// TwinCAT 3 PLC project STRIX1200
// ProgramVersion: 3.1.4024.0
// libraries:
//   CmpBitmapPool, * (System)
//   Tc2_MC2, * (Beckhoff Automation GmbH)
//   Tc2_Standard, * (Beckhoff Automation GmbH)
//   Tc2_System, * (Beckhoff Automation GmbH)
//   Tc2_Utilities, * (Beckhoff Automation GmbH)
//   Tc3_Module, * (Beckhoff Automation GmbH)
//   VisuDialogs, * (System)
// project tree:
//   / GlobalTextList.TcGTLO, PlcTask.TcTTO, Visualization Manager.TcVMO (not stored), VISU_TASK.TcTTO
//   POUs/ACTION/ E_ACTION_STATE.TcDUT, FB_ACTION.TcPOU (not stored), FB_AnalogSensor.TcPOU (not stored), vACTION.TcVIS
//   POUs/AXES/ AXES_CYCLE.TcPOU, E_AXIS_STATE.TcDUT, FB_Axis.TcPOU, GVL_AXES.TcGVL, vAXES2.TcVIS, vAXIS.TcVIS, vAXES1.TcVIS
//   POUs/EVENT_LOGGER/ E_EventType.TcDUT, FB_EventLogger.TcPOU, GVL_EVENT_LOGGER.TcGVL, ST_Event.TcDUT, UpdateEventTimestampWithSystemTime.TcPOU, UpdateTimeStamp.TcPOU, vEVENT_LOGGER.TcVIS
//   POUs/ GVL_MAIN.TcGVL (not stored), MAIN.TcPOU (not stored)
//   POUs/IOs/ sEL1809.TcDUT, sEL2809.TcDUT
//   POUs/PISTONS/ E_PISTON_STATE.TcDUT, E_PISTON_TYPE.TcDUT, FB_PISTON.TcPOU, PIST_CYCLE.TcPOU, ST_PISTON.TcDUT, vPISTONS.TcVIS, vPISTON.TcVIS
//   VISUs/VISUs/ ImagePool.TcIPO (not stored), vCOMM.TcVIS, vMAIN.TcVIS
// real-time tasks:
//   TASK PlcTask: cycle T#10ms, priority 20, ADS port 350
//   TASK VISU_TASK: cycle T#70000us, priority 30, ADS port 351
// motion (NC):
//   TASK NC-Task 1 SAF: cycle T#2ms, priority 4, ADS port 501
//   TASK NC-Task 1 SVB: cycle T#10ms, priority 8, ADS port 511
//   AXIS XY1 (id 2)
//     Dynamic: AccelerationMaximum=1500, DecelerationMaximum=1500, Acceleration=400, Deceleration=400, Jerk=40000
//     Velo: SlowManual=3, FastManual=6, Maximum=200
//     OtherSettings: AllowMotionCmdToSlave=true
//     encoder EncType=4
//       EncPara: ScaleFactorNumerator=0.001, EncMode=3, MaxCount=#xffffffff
//         TimeComp: TimeCompMode=1, EncDelayCycles=4
//     drive DrvType=5
//       Analog: VeloReferenz=200, TorqueSetpointScale=10, ScaleFactorActTorque=0.1
//       TimeComp: TimeCompMode=1, TaskDelayCycles=1
//     controller CtrType=1
//       CtrPara: PriorControlFactor=1
//         PosDiffControl: Enable=false
//         PID: PosKp=50
//         Observer: BandWidth=20
//   AXIS LIFT2 (id 3)
//     OtherSettings: AllowMotionCmdToSlave=true
//     encoder EncType=1
//     drive DrvType=5
//       Analog: TorqueSetpointScale=10, ScaleFactorActTorque=0.1
//       TimeComp: TaskDelayCycles=1
//     controller CtrType=1
//       CtrPara: PriorControlFactor=1
//         PID: PosKp=50
//         Observer: BandWidth=20
//   AXIS XY2 (id 4)
//     OtherSettings: AllowMotionCmdToSlave=true
//     encoder EncType=1
//     drive DrvType=5
//       Analog: TorqueSetpointScale=10, ScaleFactorActTorque=0.1
//       TimeComp: TaskDelayCycles=1
//     controller CtrType=1
//       CtrPara: PriorControlFactor=1
//         PID: PosKp=50
//         Observer: BandWidth=20
//   AXIS LIFT1 (id 1)
//     Dynamic: AccelerationMaximum=300, DecelerationMaximum=300, Acceleration=400, Deceleration=400, Jerk=40000
//     Velo: SlowManual=10, FastManual=30, Maximum=200
//     OtherSettings: AllowMotionCmdToSlave=true
//     encoder EncType=4
//       EncPara: ScaleFactorNumerator=0.001, EncMode=3, MaxCount=#xffffffff
//         TimeComp: TimeCompMode=1
//     drive DrvType=5
//       Analog: VeloReferenz=200, TorqueSetpointScale=10, ScaleFactorActTorque=0.1
//       TimeComp: TimeCompMode=1, TaskDelayCycles=1
//     controller CtrType=1
//       CtrPara: PriorControlFactor=1
//         PosDiffControl: Enable=false
//         PID: PosKp=50
//         Observer: BandWidth=20
// I/O:
//   DEVICE Device 1 (EtherCAT), AmsNetId 5.144.185.120.2.1
//     Term 1 (EK1100) [EK1100 EtherCAT Coupler (2A E-Bus)]
//       Term 2 (EL1809) [EL1809 16Ch. Dig. Input 24V, 3ms]
//       Term 3 (EL2809) [EL2809 16Ch. Dig. Output 24V, 0.5A]
//       Term 4 (EL2522) [EL2522 2Ch. Pulse Train Output]
//       Term 5 (EL3064) [EL3064 4Ch. Ana. Input 0-10V]
//       Term 6 (EL9011) [EL9011 End Terminal]
// variable links:
//   NC-Task 1 SAF/Axes/LIFT1 <-> Device 1 (EtherCAT)/Term 1 (EK1100)/Term 4 (EL2522)
//     Drive/Inputs/In/nDcOutputTime <-> InfoData/DcOutputShift
//     Drive/Inputs/In/nState1 @bit 6 <-> PTO Status Channel 2/Status/Error
//     Drive/Inputs/In/nState1 @bit 1 <-> PTO Status Channel 2/Status/Ramp active
//     Drive/Inputs/In/nState1 <-> PTO Status Channel 2/Status/Sel. Ack/End counter
//     Drive/Inputs/In/nState2 @bit 5 <-> PTO Status Channel 2/Status/Sync error
//     Drive/Inputs/In/nState2 @bit 7 <-> PTO Status Channel 2/Status/TxPDO Toggle
//     Drive/Inputs/In/nState4 @bit 1 <-> WcState/InputToggle
//     Drive/Inputs/In/nState4 <-> WcState/WcState
//     Drive/Outputs/Out/nCtrl1 @bit 1 <-> PTO Control Channel 2/Control/Disable ramp
//     Drive/Outputs/Out/nCtrl1 <-> PTO Control Channel 2/Control/Frequency select
//     Drive/Outputs/Out/nCtrl1 @bit 2 <-> PTO Control Channel 2/Control/Go counter
//     Drive/Outputs/Out/nDataOut1[0] <-> PTO Control Channel 2/Frequency value
//     Drive/Outputs/Out/nDataOut5 <-> PTO Target Channel 2/Target counter value
//     Enc/Inputs/In/nDataIn1 <-> ENC Status Channel 2/Counter value
//     Enc/Inputs/In/nDcInputTime <-> InfoData/DcInputShift
//     Enc/Inputs/In/nState1 @bit 4 <-> ENC Status Channel 2/Status/Counter overflow
//     Enc/Inputs/In/nState1 @bit 3 <-> ENC Status Channel 2/Status/Counter underflow
//     Enc/Inputs/In/nState1 @bit 2 <-> ENC Status Channel 2/Status/Set counter done
//     Enc/Inputs/In/nState2 @bit 5 <-> ENC Status Channel 2/Status/Sync error
//     Enc/Inputs/In/nState2 @bit 6 <-> ENC Status Channel 2/Status/TxPDO State
//     Enc/Inputs/In/nState2 @bit 7 <-> ENC Status Channel 2/Status/TxPDO Toggle
//     Enc/Inputs/In/nState4 @bit 1 <-> WcState/InputToggle
//     Enc/Inputs/In/nState4 <-> WcState/WcState
//     Enc/Outputs/Out/nCtrl1 @bit 2 <-> ENC Control Channel 2/Control/Set counter
//     Enc/Outputs/Out/nCtrl2 @bit 7 <-> ENC Control Channel 2/Control/Reserved
//     Enc/Outputs/Out/nDataOut1 <-> ENC Control Channel 2/Set counter value
//   NC-Task 1 SAF/Axes/XY1 <-> Device 1 (EtherCAT)/Term 1 (EK1100)/Term 4 (EL2522)
//     Drive/Inputs/In/nDcOutputTime <-> InfoData/DcOutputShift
//     Drive/Inputs/In/nState1 @bit 6 <-> PTO Status Channel 1/Status/Error
//     Drive/Inputs/In/nState1 @bit 1 <-> PTO Status Channel 1/Status/Ramp active
//     Drive/Inputs/In/nState1 <-> PTO Status Channel 1/Status/Sel. Ack/End counter
//     Drive/Inputs/In/nState2 @bit 5 <-> PTO Status Channel 1/Status/Sync error
//     Drive/Inputs/In/nState2 @bit 7 <-> PTO Status Channel 1/Status/TxPDO Toggle
//     Drive/Inputs/In/nState4 @bit 1 <-> WcState/InputToggle
//     Drive/Inputs/In/nState4 <-> WcState/WcState
//     Drive/Outputs/Out/nCtrl1 @bit 1 <-> PTO Control Channel 1/Control/Disable ramp
//     Drive/Outputs/Out/nCtrl1 <-> PTO Control Channel 1/Control/Frequency select
//     Drive/Outputs/Out/nCtrl1 @bit 2 <-> PTO Control Channel 1/Control/Go counter
//     Drive/Outputs/Out/nDataOut1[0] <-> PTO Control Channel 1/Frequency value
//     Drive/Outputs/Out/nDataOut5 <-> PTO Target Channel 1/Target counter value
//     Enc/Inputs/In/nDataIn1 <-> ENC Status Channel 1/Counter value
//     Enc/Inputs/In/nDcInputTime <-> InfoData/DcInputShift
//     Enc/Inputs/In/nState1 @bit 4 <-> ENC Status Channel 1/Status/Counter overflow
//     Enc/Inputs/In/nState1 @bit 3 <-> ENC Status Channel 1/Status/Counter underflow
//     Enc/Inputs/In/nState1 @bit 2 <-> ENC Status Channel 1/Status/Set counter done
//     Enc/Inputs/In/nState2 @bit 5 <-> ENC Status Channel 1/Status/Sync error
//     Enc/Inputs/In/nState2 @bit 6 <-> ENC Status Channel 1/Status/TxPDO State
//     Enc/Inputs/In/nState2 @bit 7 <-> ENC Status Channel 1/Status/TxPDO Toggle
//     Enc/Inputs/In/nState4 @bit 1 <-> WcState/InputToggle
//     Enc/Inputs/In/nState4 <-> WcState/WcState
//     Enc/Outputs/Out/nCtrl1 @bit 2 <-> ENC Control Channel 1/Control/Set counter
//     Enc/Outputs/Out/nCtrl2 @bit 7 <-> ENC Control Channel 1/Control/Reserved
//     Enc/Outputs/Out/nDataOut1 <-> ENC Control Channel 1/Set counter value
//   STRIX1200/STRIX1200 Instance <-> Device 1 (EtherCAT)/Term 1 (EK1100)/Term 2 (EL1809)
//     PlcTask Inputs/GVL_MAIN.LIFT1closedLimit <-> Channel 3/Input
//     PlcTask Inputs/GVL_MAIN.LIFT1openedLimit <-> Channel 4/Input
//     PlcTask Inputs/GVL_MAIN.PIST1closed <-> Channel 5/Input
//     PlcTask Inputs/GVL_MAIN.PIST1opened <-> Channel 6/Input
//     PlcTask Inputs/GVL_MAIN.XY1closedLimit <-> Channel 1/Input
//     PlcTask Inputs/GVL_MAIN.XY1openedLimit <-> Channel 2/Input
//   STRIX1200/STRIX1200 Instance <-> Device 1 (EtherCAT)/Term 1 (EK1100)/Term 3 (EL2809)
//     PlcTask Outputs/GVL_MAIN.CARGHERon <-> Channel 1/Output
//     PlcTask Outputs/GVL_MAIN.LED <-> Channel 6/Output
//     PlcTask Outputs/GVL_MAIN.PIST1close <-> Channel 2/Output
//     PlcTask Outputs/GVL_MAIN.PIST1open <-> Channel 3/Output
//     PlcTask Outputs/GVL_MAIN.PTCoff <-> Channel 5/Output
//     PlcTask Outputs/GVL_MAIN.PTCon <-> Channel 4/Output
//     PlcTask Outputs/GVL_MAIN.WARNING2 <-> Channel 7/Output
//     PlcTask Outputs/GVL_MAIN.bDISABLE_LIFT1 <-> Channel 14/Output
//     PlcTask Outputs/GVL_MAIN.bDISABLE_XY1 <-> Channel 15/Output
//   STRIX1200/STRIX1200 Instance <-> Device 1 (EtherCAT)/Term 1 (EK1100)/Term 5 (EL3064)
//     PlcTask Inputs/GVL_MAIN.iCURRENT_CHARGE1 <-> AI Standard Channel 2/Value
//     PlcTask Inputs/GVL_MAIN.iCURRENT_PISTON1 <-> AI Standard Channel 3/Value
//     PlcTask Inputs/GVL_MAIN.iTEMP1 <-> AI Standard Channel 4/Value
//     PlcTask Inputs/GVL_MAIN.iVOLTAGE1 <-> AI Standard Channel 1/Value
//   STRIX1200/STRIX1200 Instance <-> NC-Task 1 SAF/Axes/LIFT1
//     PlcTask Inputs/GVL_MAIN.LIFT1.Axis.NcToPlc <-> Outputs/ToPlc
//     PlcTask Outputs/GVL_MAIN.LIFT1.Axis.PlcToNc <-> Inputs/FromPlc
//   STRIX1200/STRIX1200 Instance <-> NC-Task 1 SAF/Axes/LIFT2
//     PlcTask Inputs/GVL_MAIN.LIFT2.Axis.NcToPlc <-> Outputs/ToPlc
//     PlcTask Outputs/GVL_MAIN.LIFT2.Axis.PlcToNc <-> Inputs/FromPlc
//   STRIX1200/STRIX1200 Instance <-> NC-Task 1 SAF/Axes/XY1
//     PlcTask Inputs/GVL_MAIN.XY1.Axis.NcToPlc <-> Outputs/ToPlc
//     PlcTask Outputs/GVL_MAIN.XY1.Axis.PlcToNc <-> Inputs/FromPlc
//   STRIX1200/STRIX1200 Instance <-> NC-Task 1 SAF/Axes/XY2
//     PlcTask Inputs/GVL_MAIN.XY2.Axis.NcToPlc <-> Outputs/ToPlc
//     PlcTask Outputs/GVL_MAIN.XY2.Axis.PlcToNc <-> Inputs/FromPlc

CONFIGURATION STRIX1200
    RESOURCE PLC ON TwinCAT3
        TASK PlcTask(INTERVAL := T#10ms, PRIORITY := 20);
        TASK VISU_TASK(INTERVAL := T#70000us, PRIORITY := 30);
        PROGRAM MAIN WITH PlcTask : MAIN;
        PROGRAM VisuElems_Visu_Prg WITH VISU_TASK : VisuElems.Visu_Prg;
    END_RESOURCE
END_CONFIGURATION

// ---- POUs/ACTION/E_ACTION_STATE.TcDUT
{attribute 'qualified_only'}
{attribute 'strict'}
TYPE E_ACTION_STATE :
(
	uninit := 0,
	st1,
	st2,
	st3,
	st4,
	st5,
	st6,
	st7,
	st8,
	st9,
	ready:=100,
	error:=99
);
END_TYPE

// ---- POUs/AXES/E_AXIS_STATE.TcDUT
{attribute 'qualified_only'}
{attribute 'strict'}
TYPE E_AXIS_STATE :
(
	uninit:=0,
	opening,
	open_dec,
	opened,
	closing,
	close_dec,
	closed,
	ready,
	error
);
END_TYPE

// ---- POUs/EVENT_LOGGER/E_EventType.TcDUT
{attribute 'qualified_only'}
{attribute 'strict'}
TYPE E_EventType :
(
	Alarm := 0,
	Message:=1
);
END_TYPE

// ---- POUs/EVENT_LOGGER/ST_Event.TcDUT
TYPE ST_Event :
STRUCT
	eEventType: STRING(255); 
	eEventSeverity: STRING(255);
	nEventIdentity: UDINT;
	sEventName: STRING(255);
	sEventText: STRING(255);
	dtTimestamp: DATE_AND_TIME;
	
END_STRUCT
END_TYPE

// ---- POUs/IOs/sEL1809.TcDUT
TYPE sEL1809 :
STRUCT
	ch1  :BOOL;
	ch2  :BOOL;
	ch3  :BOOL;
	ch4  :BOOL;
	ch5  :BOOL;
	ch6  :BOOL;
	ch7  :BOOL;
	ch8  :BOOL;
	ch9  :BOOL;
	ch10  :BOOL;
	ch11  :BOOL;
	ch12  :BOOL;
	ch13  :BOOL;
	ch14  :BOOL;
	ch15  :BOOL;
	ch16  :BOOL;
END_STRUCT
END_TYPE

// ---- POUs/IOs/sEL2809.TcDUT
TYPE sEL2809 :
STRUCT
	ch1  :BOOL;
	ch2  :BOOL;
	ch3  :BOOL;
	ch4  :BOOL;
	ch5  :BOOL;
	ch6  :BOOL;
	ch7  :BOOL;
	ch8  :BOOL;
	ch9  :BOOL;
	ch10  :BOOL;
	ch11  :BOOL;
	ch12  :BOOL;
	ch13  :BOOL;
	ch14  :BOOL;
	ch15  :BOOL;
	ch16  :BOOL;
END_STRUCT
END_TYPE

// ---- POUs/PISTONS/E_PISTON_STATE.TcDUT
{attribute 'qualified_only'}
{attribute 'strict'}
TYPE E_PISTON_STATE :
(
	uninit:=0,
	ready,
	opening,
	opened,
	closing,
	closed,
	error,
	ununinit
);
END_TYPE

// ---- POUs/PISTONS/E_PISTON_TYPE.TcDUT
{attribute 'qualified_only'}
{attribute 'strict'}
TYPE E_PISTON_TYPE :
(
	NO_SENSORS,
	ONLY_OPEN,
	ONLY_CLOSE,
	BOTH
);
END_TYPE

// ---- POUs/PISTONS/ST_PISTON.TcDUT
 TYPE ST_PISTON :
STRUCT
	ePISTON_TYPE: E_PISTON_TYPE;
	nNAME: STRING;
	openTime: REAL:=5;
	closeTime: REAL:=5;
	timeoutOpen:  TIME:=T#5S;
	timeoutClose: TIME:=T#5S;
	bOPEN_BY_DEFAULT: BOOL:= FALSE;
	
	
END_STRUCT
	
END_TYPE

// ---- POUs/AXES/GVL_AXES.TcGVL
//{attribute 'qualified_only'}
VAR_GLOBAL
	
	
END_VAR

// ---- POUs/EVENT_LOGGER/GVL_EVENT_LOGGER.TcGVL
//{attribute 'qualified_only'}
VAR_GLOBAL
	// ================================== error and logs ==============================
	sError:STRING;
	gEventType: STRING(255); 
	gEventSeverity: STRING(255);
	gEventIdentity: UDINT:=0;
	gEventText: STRING(255):='Startup Event';
	gEventName: STRING(255);
	sEventTime: STRING(255);
	fbEventLogger: FB_EventLogger;
	WriteLogToFile:BOOL:=FALSE;
	sLog:STRING(255);
	bBuffer_full:BOOL:=FALSE;
END_VAR

// ---- POUs/EVENT_LOGGER/FB_EventLogger.TcPOU
FUNCTION_BLOCK FB_EventLogger
VAR_INPUT
END_VAR
VAR_OUTPUT
END_VAR
VAR
	buffer_counter:INT;
	EventBuffer: ARRAY[1..MAXIMUN_SIZE_OF_EVENT_BUFFR] OF ST_Event;
	EventBuffer_clear: ARRAY[1..MAXIMUN_SIZE_OF_EVENT_BUFFR] OF ST_Event;
	EventBufferIndex:INT:=0;
END_VAR
VAR CONSTANT
	MAXIMUN_SIZE_OF_EVENT_BUFFR:INT :=100;
END_VAR

METHOD IsEventBufferFull : BOOL
VAR_INPUT
END_VAR
IF (EventBufferIndex+1) > MAXIMUN_SIZE_OF_EVENT_BUFFR THEN
	EventBuffer:=EventBuffer_clear;
	EventBufferIndex:=0 ;
	//IsEventBufferFull:=TRUE; 
END_IF
IsEventBufferFull:=FALSE;
END_METHOD

(* returns false if not succesfull*) 
METHOD PUBLIC mAdd : BOOL
VAR_INPUT
	
END_VAR

VAR
	arrDataToWrite: INT;
END_VAR

IF NOT IsEventBufferFull() THEN
	EventBufferIndex:=EventBufferIndex+1;
	EventBuffer[EventBufferIndex].eEventType:=gEventType;
	EventBuffer[EventBufferIndex].eEventSeverity:=gEventSeverity;
	EventBuffer[EventBufferIndex].nEventIdentity:=gEventIdentity;
	EventBuffer[EventBufferIndex].sEventName:=gEventName;
	EventBuffer[EventBufferIndex].sEventText:=gEventText;
	UpdateEventTimestampWithSystemTime (stEvent:=EventBuffer[EventBufferIndex]); 
	sEventTime:= DT_TO_STRING (EventBuffer[EventBufferIndex].dtTimestamp);
	mAdd:=TRUE ;
ELSE
	mAdd:=FALSE;
END_IF
END_METHOD

END_FUNCTION_BLOCK

// ---- POUs/EVENT_LOGGER/UpdateEventTimestampWithSystemTime.TcPOU
FUNCTION UpdateEventTimestampWithSystemTime 
VAR_INPUT
	stEvent: REFERENCE TO ST_Event;  
	
END_VAR
VAR
	fbGETSYSTEMTIME : GETSYSTEMTIME;
	stFileTime : T_FILETIME;
END_VAR

fbGETSYSTEMTIME(timeLoDW =>stFileTime.dwLowDateTime ,
				timeHiDW =>stFileTime.dwHighDateTime );
				
stEvent.dtTimestamp:= FILETIME_TO_DT(fileTime := stFileTime);

END_FUNCTION

// ---- POUs/AXES/AXES_CYCLE.TcPOU
PROGRAM AXES_CYCLE
VAR
END_VAR

GRP1();

ACTION GRP1:
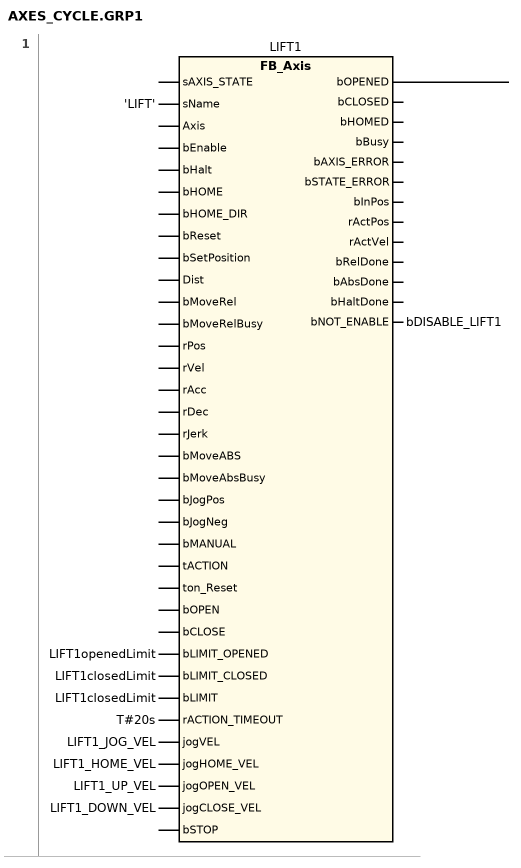
// NETWORK 1
LIFT1(
    sName := 'LIFT',
    bLIMIT_OPENED := LIFT1openedLimit,
    bLIMIT_CLOSED := LIFT1closedLimit,
    bLIMIT := LIFT1closedLimit,
    rACTION_TIMEOUT := T#20s,
    jogVEL := LIFT1_JOG_VEL,
    jogHOME_VEL := LIFT1_HOME_VEL,
    jogOPEN_VEL := LIFT1_UP_VEL,
    jogCLOSE_VEL := LIFT1_DOWN_VEL,
    bNOT_ENABLE => bDISABLE_LIFT1); // FB_Axis

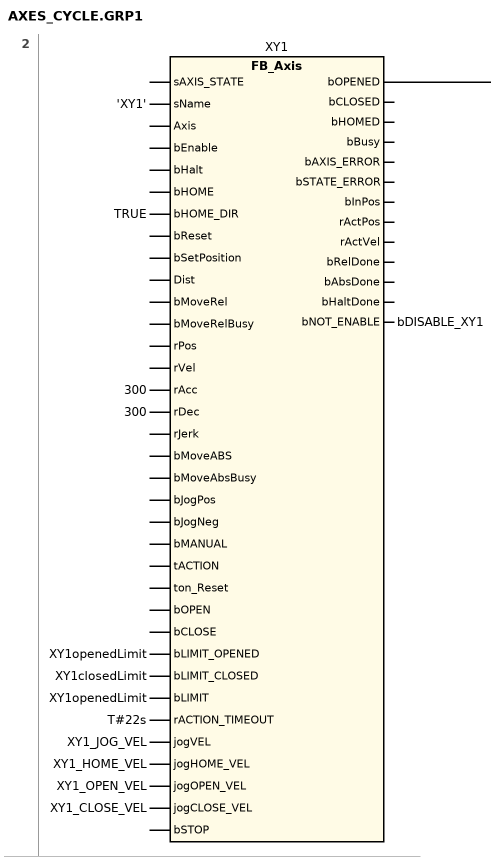
// NETWORK 2
XY1(
    sName := 'XY1',
    bHOME_DIR := TRUE,
    rAcc := 300,
    rDec := 300,
    bLIMIT_OPENED := XY1openedLimit,
    bLIMIT_CLOSED := XY1closedLimit,
    bLIMIT := XY1openedLimit,
    rACTION_TIMEOUT := T#22s,
    jogVEL := XY1_JOG_VEL,
    jogHOME_VEL := XY1_HOME_VEL,
    jogOPEN_VEL := XY1_OPEN_VEL,
    jogCLOSE_VEL := XY1_CLOSE_VEL,
    bNOT_ENABLE => bDISABLE_XY1); // FB_Axis

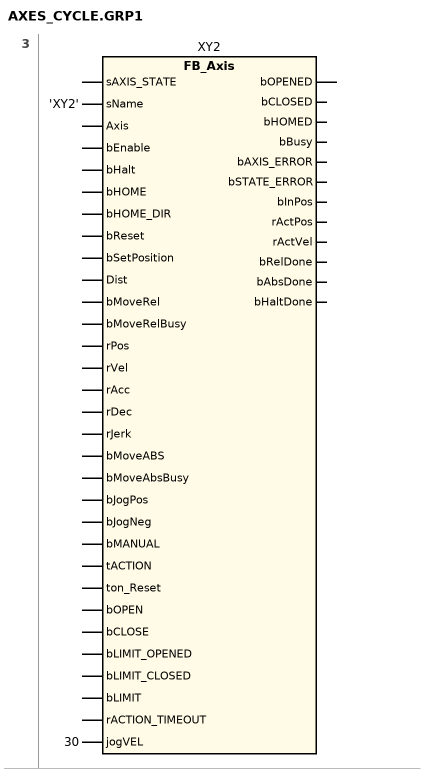
// NETWORK 3
XY2(sName := 'XY2', jogVEL := 30); // FB_Axis

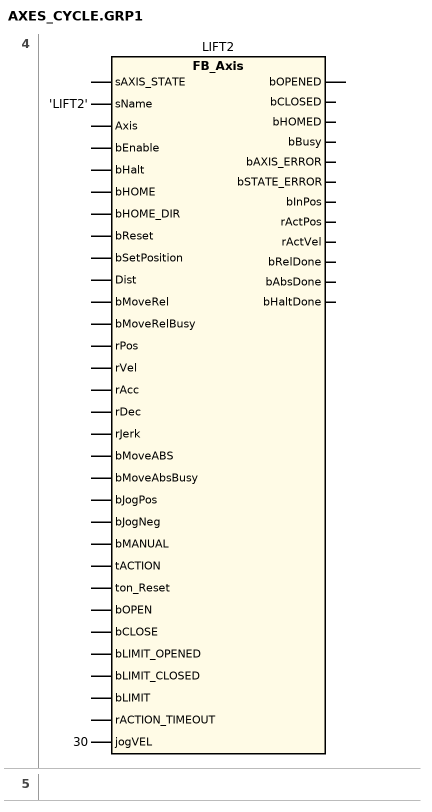
// NETWORK 4
LIFT2(sName := 'LIFT2', jogVEL := 30); // FB_Axis

// NETWORK 5
END_ACTION

END_PROGRAM

// ---- POUs/AXES/FB_Axis.TcPOU
FUNCTION_BLOCK FB_Axis
VAR_INPUT
	
	sAXIS_STATE:STRING:='UNINIT';
	sName:STRING;
	Axis:Axis_ref;
	bEnable:BOOL:=FALSE;
	bHalt:BOOL:=FALSE;
	bHOME:BOOL:=FALSE;
	bHOME_DIR:BOOL;
	bReset:BOOL:=FALSE;
	bSetPosition:BOOL:=FALSE;
	Dist:REAL;
	bMoveRel:BOOL:=FALSE;
	bMoveRelBusy:BOOL;
	rPos:LREAL;
	rVel:LREAL:=20;
	rAcc:LREAL;
	rDec:LREAL;
	rJerk:LREAL;
	bMoveABS:BOOL:=FALSE;
	bMoveAbsBusy:BOOL;
	bJogPos:BOOL;
	bJogNeg:BOOL;
	bMANUAL:BOOL:=FALSE;
	tACTION:TON;
	ton_Reset: TON;
	bOPEN:BOOL;
	bCLOSE:BOOL;
	bLIMIT_OPENED:BOOL;
	bLIMIT_CLOSED:BOOL;
	bLIMIT:BOOL;
	rACTION_TIMEOUT:TIME:=T#10S;
	jogVEL: REAL;
	jogHOME_VEL: REAL;
	jogOPEN_VEL: REAL;
	jogCLOSE_VEL: REAL;
	bSTOP:BOOL;
	bSTOP_ALL:BOOL;
END_VAR

VAR_OUTPUT
	bOPENED:BOOL;
	bCLOSED:BOOL;
	bHOMED:BOOL;
	bBusy: BOOL;
	bAXIS_ERROR:BOOL;
	bSTATE_ERROR:BOOL;
	bInPos:BOOL;
	rActPos:LREAL;
	rActVel:LREAL;
	bRelDone:BOOL;
	bAbsDone:BOOL;
	bHaltDone:BOOL;
	bNOT_ENABLE:BOOL;
END_VAR
VAR
	bSTART_ACTION:BOOL;
	iHOME_STATE: INT:=98;
	iAXIS_STATE:INT:=98;
	tDelay: TON;
	bDelay:BOOL:=FALSE;
	MoveAbsolute: MC_MoveAbsolute;
	power: MC_Power;
	Reset: MC_Reset;
	SetPosition: MC_SetPosition;
	JOG: MC_Jog;
	RELATIVE: MC_MoveRelative;
	HALT: MC_Halt;
	HOME: MC_Home;
	bFirst_run:BOOL:=FALSE;
	bStopBusy:BOOL;
	
	
	
	
END_VAR

IF NOT bFirst_run THEN
	RESET.Execute:=TRUE;
	 bFirst_run:=TRUE;
END_IF
bNOT_ENABLE:=NOT bENABLE;
rActPos:=Axis.NcToPlc.ActPos;
rActVel:=Axis.NcToPlc.ActVelo;



IF RELATIVE.Busy OR JOG.Busy OR moveAbsolute.busy THEN
	bBusy:=TRUE;
	bHOMED:=FALSE;
END_IF
IF NOT RELATIVE.Busy AND NOT JOG.Busy AND NOT moveAbsolute.busy THEN
	bBusy:=FALSE;
END_IF

IF POWER.error OR RELATIVE.error OR MoveAbsolute.error OR JOG.error THEN
	bAXIS_ERROR:=TRUE;
END_IF
IF NOT POWER.error AND NOT RELATIVE.error AND NOT MoveAbsolute.error AND NOT JOG.error THEN
	bAXIS_ERROR:=FALSE;
END_IF

IF bRelDone OR  bAbsDone THEN
	bInPos:=TRUE;
END_IF
IF bBusy THEN
	bInPos:=FALSE;
	bRelDone:=FALSE;
	bAbsDone:=FALSE;
END_IF


CMDs();
mAXIS_STATE_MACHINE();

ACTION aAXIS_ERROR:
gEventType:= 'axis Alarm'; 
gEventSeverity:= 'Error';

gEventName:= sNAME;
IF iAXIS_STATE=1  THEN
	gEventText:='axis homing';
	gEventIdentity:=2001;
END_IF
IF iAXIS_STATE=20  THEN
	gEventText:='axis opening';
	gEventIdentity:=2002;
END_IF
IF iAXIS_STATE=40  THEN
	gEventText:='axis closing';
	gEventIdentity:=2003;
END_IF
fbEventLogger.mAdd();
END_ACTION

METHOD clear_cmd_req : BOOL
VAR_INPUT
END_VAR

bMoveABS:= bMoveRel:= bJogPos:= bJogNeg:=FALSE;
END_METHOD

ACTION CMDs:
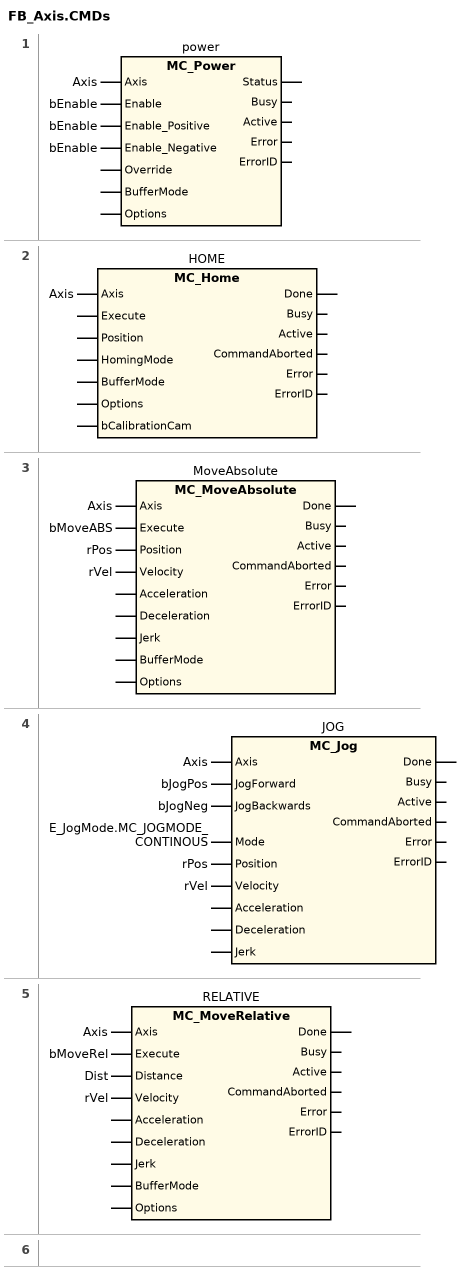
// NETWORK 1
power(Axis := Axis, Enable := bEnable, Enable_Positive := bEnable, Enable_Negative := bEnable); // MC_Power

// NETWORK 2
HOME(Axis := Axis); // MC_Home

// NETWORK 3
MoveAbsolute(Axis := Axis, Execute := bMoveABS, Position := rPos, Velocity := rVel); // MC_MoveAbsolute

// NETWORK 4
JOG(
    Axis := Axis,
    JogForward := bJogPos,
    JogBackwards := bJogNeg,
    Mode := E_JogMode.MC_JOGMODE_CONTINOUS,
    Position := rPos,
    Velocity := rVel); // MC_Jog

// NETWORK 5
RELATIVE(Axis := Axis, Execute := bMoveRel, Distance := Dist, Velocity := rVel); // MC_MoveRelative

// NETWORK 6

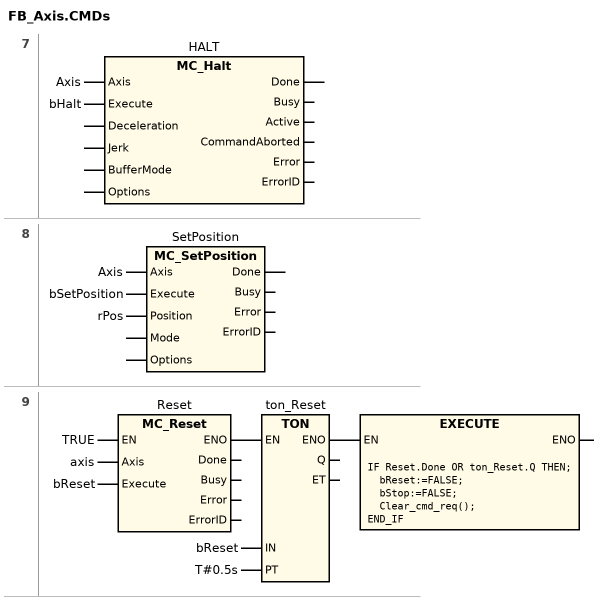
// NETWORK 7
HALT(Axis := Axis, Execute := bHalt); // MC_Halt

// NETWORK 8
SetPosition(Axis := Axis, Execute := bSetPosition, Position := rPos); // MC_SetPosition

// NETWORK 9
Reset(Axis := axis, Execute := bReset); // MC_Reset
ton_Reset(IN := bReset, PT := T#0.5s); // TON

IF Reset.Done OR ton_Reset.Q THEN;
	bReset:=FALSE;
	bStop:=FALSE;
	Clear_cmd_req();
END_IF
END_ACTION

METHOD mAXIS_STATE_MACHINE : BOOL
VAR_INPUT
	
END_VAR
tACTION(IN:= bSTART_ACTION, PT:=rACTION_TIMEOUT , Q=> , ET=> );
IF bHOME_DIR THEN
	bLIMIT:=bLIMIT_OPENED;
ELSE
	bLIMIT:=bLIMIT_CLOSED;
END_IF

IF bSTOP_ALL THEN
	iAXIS_STATE:=99;
	bSTOP_ALL:=FALSE;
	bSTART_ACTION:=FALSE;
END_IF

CASE iAXIS_STATE OF
	1:// ============================================== HOMING
		bSTART_ACTION:=TRUE;
		sAXIS_STATE:='HOMING - TO SENSOR';
		bOPENED:=FALSE;bCLOSED:=FALSE;bOPEN:=FALSE;bCLOSE:=FALSE;bHOMED:=FALSE;bHOME:=FALSE;
		bENABLE:=TRUE;
		rVel:= jogHOME_VEL;
		IF bHOME_DIR THEN
			bJogPos:=TRUE;
		ELSE
			bJogNeg:=TRUE;
		END_IF
		
		IF bLIMIT THEN
			bSTART_ACTION:=FALSE;
			bJogNeg:=FALSE;
			bJogPos:=FALSE;
			iAXIS_STATE:=2;
		END_IF
		IF tACTION.Q THEN
			bSTART_ACTION:=FALSE;
			aAXIS_ERROR();
			iAXIS_STATE:=99;
			bSTATE_ERROR:=TRUE;
		END_IF
	2://FROM LIMIT
			sAXIS_STATE:= 'HOMING- FROM SENSOR';
			IF Axis.NcToPlc.ActVelo= 0 THEN
				
				//rVel:= 3;
				//IF bHOME_DIR THEN
				//	bJogNeg:=TRUE;
				//ELSE
					//bJogPos:=TRUE;
				//END_IF
				iAXIS_STATE:=3;
			END_IF	
	3:// FINISH
			//IF NOT bLIMIT THEN
				//bJogNeg:=FALSE;
				//bJogPos:=FALSE;
				IF Axis.NcToPlc.ActVelo= 0 THEN
					bHOMED:=TRUE;
					IF bHOME_DIR THEN
						iAXIS_STATE:=100;// to ready state
						bOPENED:=TRUE;
					ELSE
						iAXIS_STATE:=100;// to ready state
						bCLOSED:=TRUE;
					END_IF
				END_IF
			//END_IF
	20://=============================================== OPENING
		sAXIS_STATE:= 'OPENING';
		bSTART_ACTION:=TRUE;
		bOPENED:=FALSE;bCLOSED:=FALSE;bOPEN:=FALSE;bCLOSE:=FALSE;bHOMED:=FALSE;bHOME:=FALSE;
		bENABLE:=TRUE;
		rVel:= jogOPEN_VEL;
		bJogPos:=TRUE;
		IF bLIMIT_OPENED THEN
			iAXIS_STATE:=21;// to deccell
			bJogPos:=FALSE;
			bSTART_ACTION:=FALSE;
		END_IF
		IF tACTION.Q THEN
			bSTART_ACTION:=FALSE;
			aAXIS_ERROR();
			iAXIS_STATE:=99;
			bSTATE_ERROR:=TRUE;
		END_IF
		
		21:
			sAXIS_STATE:= 'OPEN DECCELERATING';
			IF Axis.NcToPlc.ActVelo=0 THEN
				bENABLE:=FALSE;//////////////////////
				iAXIS_STATE:=100;
				bOPENED:=TRUE;
			END_IF
	
	40://=============================================== CLOSING
		sAXIS_STATE:= 'CLOSING';
		bSTART_ACTION:=TRUE;
		bOPENED:=FALSE;bCLOSED:=FALSE;bOPEN:=FALSE;bCLOSE:=FALSE;bHOMED:=FALSE;bHOME:=FALSE;
		bENABLE:=TRUE;
		rVel:= jogCLOSE_VEL;
		bJogNeg:=TRUE;
		IF bLIMIT_CLOSED THEN
			iAXIS_STATE:=41;// to deccell
			bJogNeg:=FALSE;
			bSTART_ACTION:=FALSE;
		END_IF
		IF tACTION.Q THEN
			bSTART_ACTION:=FALSE;
			aAXIS_ERROR();
			iAXIS_STATE:=99;
			bSTATE_ERROR:=TRUE;
		END_IF
		
		41:
			sAXIS_STATE:= 'CLOSE DECCELERATING';
			IF Axis.NcToPlc.ActVelo=0 THEN
				bENABLE:=FALSE;//////////////////////
				iAXIS_STATE:=100;
				bCLOSED:=TRUE;
			END_IF
	
	50:	//========================ABSOLUTE=====================
	sAXIS_STATE:='MOVING ABSOLUTE';
	bAbsDone:=FALSE; bOPENED:=FALSE;bCLOSED:=FALSE;bOPEN:=FALSE;bCLOSE:=FALSE;bHOMED:=FALSE;bHOME:=FALSE;
	IF moveAbsolute.Done OR HALT.Done THEN
		iAXIS_STATE:=100;
		bAbsDone:=TRUE;
		bMoveAbs:=FALSE;
	END_IF
	51://========================RELATIVE=====================
	sAXIS_STATE:='MOVING RELATIVE';
	bRelDone:=FALSE; bOPENED:=FALSE;bCLOSED:=FALSE;bOPEN:=FALSE;bCLOSE:=FALSE;bHOMED:=FALSE;bHOME:=FALSE;
	IF RELATIVE.Done OR HALT.Done THEN
		iAXIS_STATE:=100; 
		bRelDone:=TRUE;
		bMoveRel:=FALSE;
	END_IF
	52://======================= HALT =========================
	sAXIS_STATE:='HALTING';
	bHaltDone:=FALSE;bOPENED:=FALSE;bCLOSED:=FALSE;bOPEN:=FALSE;bCLOSE:=FALSE;bHOMED:=FALSE;bHOME:=FALSE;
	IF HALT.Done THEN
		iAXIS_STATE:=100;
		bHaltDone:=TRUE;
		bHALT:=FALSE;
	END_IF		
	98:// ============================================ UNINIT
		sAXIS_STATE:='UNINIT';
		IF bHOME THEN
			iAXIS_STATE:=1;
			bSTATE_ERROR:=FALSE;
		END_IF
		
	99://======================================= ERROR 
		sAXIS_STATE:='AXIS STATE ERROR';
		bJogNeg:=FALSE;
		bJogPos:=FALSE;
		bHOMED:=FALSE;
		clear_cmd_req();
		IF bHOME THEN
			iAXIS_STATE:=1;
			bSTATE_ERROR:=FALSE;
		END_IF
		
	100://=============================================== READY
		sAXIS_STATE:='READY';
		IF bOPENED THEN
		sAXIS_STATE:= 'OPENED';
		END_IF
		IF bCLOSED THEN
		sAXIS_STATE:= 'CLOSED';
		END_IF
		IF bHOME AND NOT bHOMED THEN
			iAXIS_STATE:=1;
			bSTATE_ERROR:=FALSE;
		END_IF
		IF bCLOSE AND NOT bCLOSED THEN
			iAXIS_STATE:=40;
			bSTATE_ERROR:=FALSE;
		END_IF
		IF bOPEN AND NOT bOPENED THEN
			iAXIS_STATE:=20;
			bSTATE_ERROR:=FALSE;
		END_IF
		IF bMoveAbs THEN
			iAXIS_STATE:=50;
			bSTATE_ERROR:=FALSE;
		END_IF
		IF bMoveRel THEN
			iAXIS_STATE:=51;
			bSTATE_ERROR:=FALSE;
		END_IF
		IF bHALT THEN
			iAXIS_STATE:=52;
			bSTATE_ERROR:=FALSE;
		END_IF
	
END_CASE
END_METHOD

END_FUNCTION_BLOCK

// ---- POUs/EVENT_LOGGER/UpdateTimeStamp.TcPOU
FUNCTION UpdateTimeStamp 
VAR_INPUT
	stUser : REFERENCE TO ST_USER;
END_VAR
VAR
	fbGETSYSTEMTIME : GETSYSTEMTIME;
	
	stFileTime : T_FILETIME;
END_VAR


fbGETSYSTEMTIME(timeLoDW =>stFileTime.dwLowDateTime ,
				timeHiDW =>stFileTime.dwHighDateTime );
				
stUser.dtTIME_STAMP:= FILETIME_TO_DT(fileTime := stFileTime);

END_FUNCTION

// ---- POUs/PISTONS/FB_PISTON.TcPOU
FUNCTION_BLOCK FB_PISTON
VAR_INPUT
	sSTATE:STRING:='UNINIT';
	sNAME:STRING;
	bLOCAL_MANUAL: BOOL:=FALSE;
	pist_TYPE: E_PISTON_TYPE;
	pist_STATE: E_PISTON_STATE:=E_PISTON_STATE.ununinit;
	rOPEN_TIME: TIME;
	rCLOSE_TIME: TIME;
	rOPEN_TIMEOUT: TIME;
	tCLOSE_TIMEOUT: TIME;
	bOPEN_LIMIT: BOOL;
	bCLOSED_LIMIT: BOOL;
	bOPEN_CMD: BOOL;
	bCLOSE_CMD: BOOL;
	bOPEN_SWR: BOOL;
	bCLOSE_SWR: BOOL;
	bCONDITION: BOOL:=TRUE;
	bLOCAL_RESET:BOOL;
	bHOME_FIRST: BOOL:=FALSE;
	bSTOP_ALL:BOOL:=FALSE;
	bEXTRA:BOOL:=FALSE;
	bLIFT_DOWN:BOOL;
END_VAR
VAR_OUTPUT
	bOPEN_VALVE: BOOL;
	bCLOSE_VALVE: BOOL;
	bBUSY:BOOL;
	bOPENED:BOOL;
	bCLOSED:BOOL;
	bERROR:BOOL:=FALSE;
END_VAR
VAR
	T_EXTRA: TON;
	T_OPEN: TON;
	T_OPEN_TIMEOUT: TON;
	T_CLOSE: TON;
	T_CLOSE_TIMEOUT: TON;
	bOPEN_DEFAULT: BOOL:=FALSE;
	bFIRST_DONE: BOOL:=FALSE;
	bHOMED_FIRST:BOOL:=FALSE;
END_VAR

T_OPEN(IN:= bOPEN_CMD, PT:=rOPEN_TIME , Q=> , ET=> );
T_CLOSE(IN:=  NOT bOPEN_CMD, PT:=rCLOSE_TIME , Q=> , ET=> );
T_OPEN_TIMEOUT(IN:= bOPEN_CMD , PT:= rOPEN_TIMEOUT, Q=> , ET=> );
T_CLOSE_TIMEOUT(IN:=  NOT bOPEN_CMD , PT:= tCLOSE_TIMEOUT, Q=> , ET=> );
T_EXTRA(IN:= bEXTRA, PT:=T#2S);


IF bSTOP_ALL  THEN//======================================== STOP ========
	pist_STATE:=E_PISTON_STATE.error;
	bSTOP_ALL:=FALSE;
END_IF

IF bLOCAL_RESET THEN//========================== RESET================
	bERROR:=FALSE;
	bEXTRA:=FALSE;
	bLOCAL_RESET:=FALSE;
	pist_STATE:=E_PISTON_STATE.uninit;
END_IF

IF NOT bLOCAL_MANUAL THEN//====================== MANUAL ==============
	bOPEN_CMD:=bOPEN_SWR;
END_IF



//IF bHOME_FIRST AND NOT bHOMED_FIRST THEN
	//bHOMED_FIRST:=TRUE;
	//pist_STATE:=E_PISTON_STATE.uninit;
	//bFIRST_DONE:=FALSE;//to set command to false to zero timer
//END_IF

IF NOT bFIRST_DONE THEN  // ============== check default mode ===============
	bFIRST_DONE:=TRUE;
	IF bOPEN_DEFAULT THEN
		bOPEN_CMD:=TRUE;
	ELSE
		bOPEN_CMD:=FALSE;
	END_IF
END_IF
//================================================== UNINIT =====================================================
CASE pist_STATE OF
	E_PISTON_STATE.uninit:
		bERROR:=FALSE;
		//IF bHOME_FIRST THEN
			IF bOPEN_CMD  THEN
				bOPEN_VALVE:=TRUE;
				bCLOSE_VALVE:=FALSE;
				pist_STATE:=E_PISTON_STATE.opening;
			ELSE
				bOPEN_VALVE:=FALSE;
				bCLOSE_VALVE:=TRUE;
				pist_STATE:=E_PISTON_STATE.closing;
			END_IF
		//END_IF
//================================================== OPENING =====================================================
	E_PISTON_STATE.opening:
	sSTATE:='OPENING';
	bBUSY:=TRUE; bOPENED:=FALSE; bCLOSED:=FALSE;
	CASE pist_TYPE OF//------------------------------no sensors
		E_PISTON_TYPE.NO_SENSORS:
		IF T_OPEN.Q THEN
			bOPEN_VALVE:=FALSE;
			pist_STATE:=E_PISTON_STATE.opened;
		END_IF
		//----------------------------- both sensors
		E_PISTON_TYPE.BOTH:
		IF bOPEN_LIMIT THEN
			bOPEN_VALVE:=FALSE;
			pist_STATE:=E_PISTON_STATE.opened;
		END_IF
		IF T_OPEN_TIMEOUT.Q THEN
			bOPEN_CMD:=FALSE;
			aPISTON_ERROR();
			pist_STATE:=E_PISTON_STATE.error;
		END_IF
		//----------------------------- only open sensor
		E_PISTON_TYPE.ONLY_OPEN:
		IF bOPEN_LIMIT THEN
			pist_STATE:=E_PISTON_STATE.opened;
		END_IF
		IF T_OPEN_TIMEOUT.Q THEN
			bOPEN_CMD:=FALSE;
			aPISTON_ERROR();
			pist_STATE:=E_PISTON_STATE.error;
		END_IF
		//----------------------------- only close sensor
		E_PISTON_TYPE.ONLY_CLOSE:
		IF T_OPEN.Q THEN
			pist_STATE:=E_PISTON_STATE.opened;
		END_IF
	END_CASE
//================================================== CLOSING =====================================================	
	E_PISTON_STATE.closing:
	sSTATE:='CLOSING'; bOPENED:=FALSE; bCLOSED:=FALSE;
	bBUSY:=TRUE;
	CASE pist_TYPE OF//--------------------------------------- no sensors
		E_PISTON_TYPE.NO_SENSORS:
		IF T_CLOSE.Q THEN
			pist_STATE:=E_PISTON_STATE.closed;
			bCLOSE_VALVE:=FALSE;
		END_IF
		//-------------------------------------- both sensors
		E_PISTON_TYPE.BOTH:
		IF bCLOSED_LIMIT THEN
			bEXTRA:=TRUE;
			IF T_EXTRA.Q THEN
				pist_STATE:=E_PISTON_STATE.closed;
				bCLOSE_VALVE:=FALSE;
				bEXTRA:=FALSE;
			END_IF
		ELSIF T_CLOSE_TIMEOUT.Q THEN
			bOPEN_CMD:=TRUE;
			pist_STATE:=E_PISTON_STATE.error;
			
		END_IF
		//-------------------------------------- only close sensor
		E_PISTON_TYPE.ONLY_CLOSE:
		IF bCLOSED_LIMIT THEN
			pist_STATE:=E_PISTON_STATE.closed;
		END_IF
		IF T_CLOSE_TIMEOUT.Q THEN
			bOPEN_CMD:=TRUE;
			aPISTON_ERROR();
			pist_STATE:=E_PISTON_STATE.error;
		END_IF
		//----------------------------- only close sensor
		E_PISTON_TYPE.ONLY_OPEN:
		IF T_CLOSE.Q THEN
			pist_STATE:=E_PISTON_STATE.closed;
		END_IF
	END_CASE
//================================================== OPENED =====================================================	
	E_PISTON_STATE.opened:
	sSTATE:='OPENED';
	bOPEN_VALVE:=FALSE;
	bBUSY:=FALSE; bOPENED:=TRUE; bCLOSED:=FALSE;
	IF NOT bOPEN_CMD AND  bLIFT_DOWN THEN
		pist_STATE:=E_PISTON_STATE.closing;
		bOPEN_VALVE:=FALSE;
		bCLOSE_VALVE:=TRUE;
	END_IF
	CASE pist_TYPE OF
		//-------------------------------------- both sensors
		E_PISTON_TYPE.BOTH:
		IF NOT bOPEN_LIMIT THEN
			//bOPEN_CMD:=FALSE;
			//aPISTON_ERROR();
			//pist_STATE:=E_PISTON_STATE.error;
		END_IF
		//-------------------------------------- only open sensor
		E_PISTON_TYPE.ONLY_OPEN:
		IF NOT bOPEN_LIMIT THEN
			bOPEN_CMD:=FALSE;
			aPISTON_ERROR();
			pist_STATE:=E_PISTON_STATE.error;
		END_IF
	END_CASE
//================================================== CLOSED =====================================================	
	E_PISTON_STATE.closed:
	sSTATE:='CLOSED';
	bCLOSE_VALVE:=FALSE;
	bBUSY:=FALSE; bOPENED:=FALSE; bCLOSED:=TRUE;
	IF bOPEN_CMD  THEN
		pist_STATE:=E_PISTON_STATE.opening;
		bOPEN_VALVE:=TRUE;
		bCLOSE_VALVE:=FALSE;
	END_IF
	CASE pist_TYPE OF
		//-------------------------------------- both sensors
		E_PISTON_TYPE.BOTH:
		IF NOT bCLOSED_LIMIT THEN
			bOPEN_CMD:=TRUE;
			aPISTON_ERROR();
			pist_STATE:=E_PISTON_STATE.error;
		END_IF
		//-------------------------------------- only close sensor
		E_PISTON_TYPE.ONLY_CLOSE:
		IF NOT bCLOSED_LIMIT THEN
			bOPEN_CMD:=TRUE;
			aPISTON_ERROR();
			pist_STATE:=E_PISTON_STATE.error;
		END_IF
	END_CASE
//================================================== ERROR =====================================================	
	E_PISTON_STATE.error:
	sSTATE:='ERROR';
	bERROR:=TRUE;
	bCLOSE_VALVE:=FALSE;
	bOPEN_VALVE:=FALSE;
	bEXTRA:=FALSE;
	//
END_CASE

ACTION aPISTON_ERROR:
gEventType:= 'piston Alarm'; 
gEventSeverity:= 'Error';

gEventName:= sNAME;
IF pist_STATE=E_PISTON_STATE.opening  THEN
	gEventText:='piston opening';
	gEventIdentity:=1001;
END_IF
IF pist_STATE=E_PISTON_STATE.closing THEN
	gEventText:='piston closing';
	gEventIdentity:=1002;
END_IF
IF pist_STATE=E_PISTON_STATE.closed THEN
	gEventText:='piston closed';
	gEventIdentity:=1003;
END_IF
IF pist_STATE=E_PISTON_STATE.opened THEN
	gEventText:='piston opened';
	gEventIdentity:=1004;
END_IF
fbEventLogger.mAdd();
END_ACTION

END_FUNCTION_BLOCK

// ---- POUs/PISTONS/PIST_CYCLE.TcPOU
PROGRAM PIST_CYCLE
VAR
	bFirstRun:BOOL:=FALSE;
	counter :INT;
END_VAR


//IF NOT bFirstRun THEN
//	FOR counter:=1 TO iNUMBER_OF_PISTONS BY 1 DO
//		fbPist[counter].bInit:=1;
//	END_FOR;
//bFirstRun:=TRUE;
//END_IF
 

grp1();

ACTION grp1:
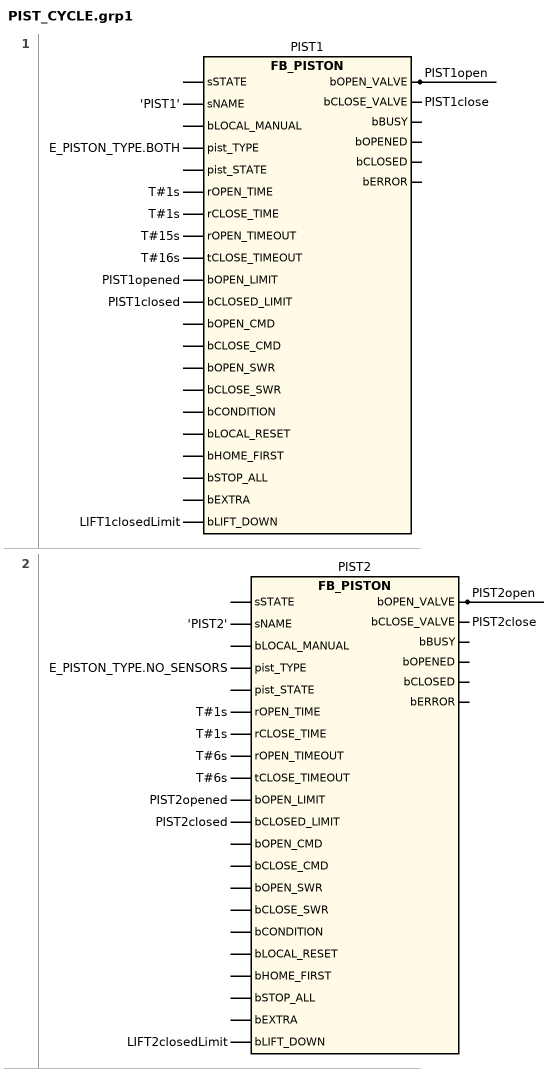
// NETWORK 1
PIST1(
    sNAME := 'PIST1',
    pist_TYPE := E_PISTON_TYPE.BOTH,
    rOPEN_TIME := T#1s,
    rCLOSE_TIME := T#1s,
    rOPEN_TIMEOUT := T#15s,
    tCLOSE_TIMEOUT := T#16s,
    bOPEN_LIMIT := PIST1opened,
    bCLOSED_LIMIT := PIST1closed,
    bLIFT_DOWN := LIFT1closedLimit,
    bOPEN_VALVE => PIST1open,
    bCLOSE_VALVE => PIST1close); // FB_PISTON

// NETWORK 2
PIST2(
    sNAME := 'PIST2',
    pist_TYPE := E_PISTON_TYPE.NO_SENSORS,
    rOPEN_TIME := T#1s,
    rCLOSE_TIME := T#1s,
    rOPEN_TIMEOUT := T#6s,
    tCLOSE_TIMEOUT := T#6s,
    bOPEN_LIMIT := PIST2opened,
    bCLOSED_LIMIT := PIST2closed,
    bLIFT_DOWN := LIFT2closedLimit,
    bOPEN_VALVE => PIST2open,
    bCLOSE_VALVE => PIST2close); // FB_PISTON
END_ACTION

END_PROGRAM

// ---- GlobalTextList.TcGTLO
TEXTLIST GlobalTextList
  450 = '%.2f'
  82 = '%.3f'
  199 = '%d'
  55 = '%f'
  571 = '%f.2'
  731 = '%f2'
  952 = '%s'
  286 = 'A1 MANUAL'
  41 = 'A:'
  396 = 'ACC'
  267 = 'Actions'
  361 = 'AENT:'
  822 = 'anualLIMIT'
  188 = 'BUSY'
  729 = 'CHARGER'
  784 = 'CHARGER ON'
  997 = 'CLOSE'
  513 = 'CLOSE ALL'
  608 = 'CLOSE VEL'
  307 = 'CLOSE XY VEL'
  293 = 'CLOSED LIMIT'
  986 = 'COOLING'
  116 = 'current'
  159 = 'CURRENT:'
  570 = 'CURRENT:[A]'
  965 = 'current[A]'
  446 = 'DIST'
  831 = 'DOWN VEL'
  904 = 'ENABLE'
  50 = 'ERROR'
  234 = 'Error Logs'
  135 = 'FAN'
  91 = 'FAN ON/OFF'
  288 = 'GO ABS'
  776 = 'GO REL'
  373 = 'HALT'
  598 = 'HOME'
  825 = 'HOME_ALL'
  512 = 'INPOS'
  837 = 'JERK'
  268 = 'JOG +'
  202 = 'JOG -'
  668 = 'LIMIT AMP'
  617 = 'LIMIT AMP:'
  251 = 'LIMIT AMP: [A]'
  412 = 'MANUAL'
  51 = 'manual'
  615 = 'Motors1'
  431 = 'Motors2'
  287 = 'OFFSET'
  189 = 'OPEN'
  149 = 'OPEN ALL'
  347 = 'OPEN VEL'
  725 = 'OPEN XY VEL'
  299 = 'OPENED LIMIT'
  920 = 'PISTON 1'
  309 = 'PISTON 2'
  419 = 'Pistons'
  100 = 'PISTONS'
  425 = 'POS'
  390 = 'Pos: %.2f'
  563 = 'POWER'
  355 = 'PTC ON'
  945 = 'PTC ON/OFF'
  507 = 'R'
  779 = 'RESET'
  68 = 'S1 MANUAL'
  89 = 'S2 MANUAL'
  830 = 'SET'
  707 = 'STOP !!'
  627 = 'SYS1'
  178 = 'SYS2'
  667 = 'System 1'
  12 = 'System 2'
  388 = 'SYSTEM 2'
  826 = 'System1'
  963 = 'System2'
  745 = 'TECHNITIAN'
  348 = 'Technitian'
  83 = 'TEMP'
  256 = 'TEMP:'
  464 = 'TEMP:[c]'
  973 = 'UP VEL'
  401 = 'V:'
  964 = 'VEL'
  60 = 'Vel: %.2f'
  888 = 'vo'
  567 = 'voltage [V]'
  291 = 'VOLTAGE:'
END_TEXTLIST

// ---- POUs/ACTION/vACTION.TcVIS
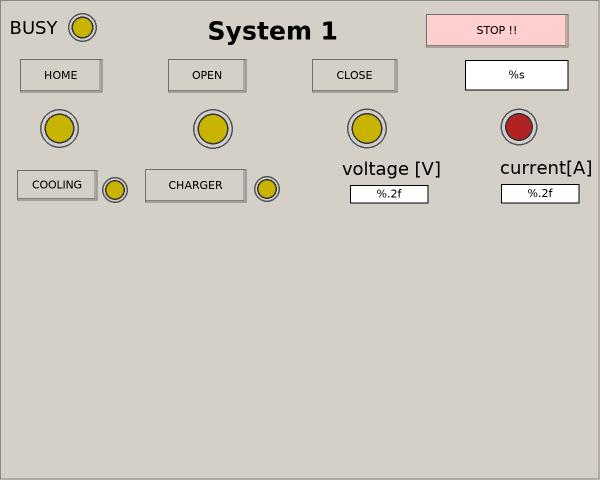
VISUALIZATION vACTION  // 600x480
VAR_IN_OUT
	vACTION:FB_ACTION;
	vACTION2:FB_ACTION;
END_VAR
    Button (20,59 82x33), "HOME", input disabled if: vACTION.bBUSY
        OnMouseDown: execute { vACTION.bHOME_ALL:=TRUE; }
    Lamp1 (37,103 45x51), variable: vACTION.bALL_HOMED, style: Lamp-Lamp1-Yellow
    Button (168,59 78x33), "OPEN", input disabled if: vACTION.bSAFE_MODE
        OnMouseDown: execute { vACTION.bOPEN_ALL:=TRUE; }
    Lamp1 (190,103 46x52), variable: vACTION.bALL_OPENED, style: Lamp-Lamp1-Yellow
    Button (312,59 85x33), "CLOSE", input disabled if: vACTION.bSAFE_MODE
        OnMouseDown: execute { vACTION.bCLOSE_ALL:=TRUE; }
    Lamp1 (344,103 46x51), variable: vACTION.bALL_CLOSED, style: Lamp-Lamp1-Yellow
    Lamp1 (498,104 42x46), variable: vACTION.bACTION_ERROR, style: Lamp-Lamp1-Red
    Rectangle (465,60 103x30), "%s", text variable: vACTION.sACTION_STATE
    Label (198,17 150x27), "System 1"
    Button (20,288 82x33), "HOME"
        OnMouseDown: execute { vACTION2.bHOME_ALL:=TRUE; }
    Lamp1 (37,332 45x51), variable: vACTION2.bALL_HOMED, style: Lamp-Lamp1-Yellow
    Button (168,288 78x33), "OPEN"
        OnMouseDown: execute { vACTION2.bOPEN_ALL:=TRUE; }
    Lamp1 (190,332 46x52), variable: vACTION2.bALL_OPENED, style: Lamp-Lamp1-Yellow
    Button (312,288 85x33), "CLOSE"
        OnMouseDown: execute { vACTION2.bCLOSE_ALL:=TRUE; }
    Lamp1 (344,332 46x51), variable: vACTION2.bALL_CLOSED, style: Lamp-Lamp1-Yellow
    Lamp1 (498,333 42x46), variable: vACTION2.bACTION_ERROR, style: Lamp-Lamp1-Red
    Rectangle (465,289 103x30), "%s", text variable: vACTION2.sACTION_STATE
    Label (121,252 150x30), "System 2"
    Button (145,169 101x33), "CHARGER"
        toggle vACTION.bCHARGE
    Rectangle (350,185 78x18), "%.2f", text variable: vACTION.iVOLTAGE_SHOW
    Label (339,155 105x28), "voltage [V]"
    Lamp1 (252,171 30x36), variable: vACTION.bCHARGE, style: Lamp-Lamp1-Yellow
    Button (16,391 101x33), "CHARGER ON"
        toggle vACTION2.bCHARGE
    Rectangle (286,391 103x30), "%f", text variable: vACTION2.iVOLTAGE_SHOW
    Label (155,396 150x30), "VOLTAGE:"
    Lamp1 (127,393 30x36), variable: vACTION2.bCHARGE, style: Lamp-Lamp1-Yellow
    Button (426,14 142x33), "STOP !!"
        OnMouseDown: execute { vACTION.bSTOP_ALL:=TRUE; }
    Button (428,249 140x33), "STOP !!"
        OnMouseDown: execute { vACTION.bSTOP_ALL:=TRUE; }
    Rectangle (7,240 571x227), invisible if: bSECOND_SYS
    Lamp1 (66,10 33x35), variable: LED, style: Lamp-Lamp1-Yellow
    Label (-5,13 77x30), "BUSY"
    Label (498,153 97x30), "current[A]"
    Rectangle (501,184 78x19), "%.2f", text variable: vACTION.iCURRENT_CHARGE_SHOW
    Button (17,170 80x30), "COOLING"
        toggle ACTION1.bPTC_ON
    Lamp1 (100,172 30x36), variable: PTCon, style: Lamp-Lamp1-Yellow
END_VISUALIZATION

// ---- POUs/AXES/vAXES2.TcVIS
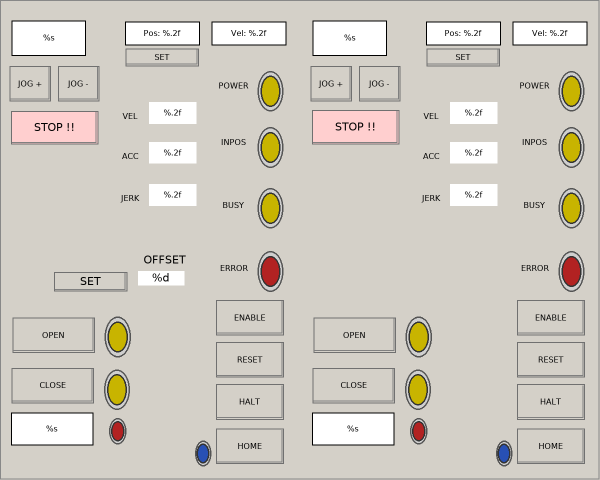
VISUALIZATION vAXES2  // 600x480
    Frame (0,3 298x468)
        shows vAXIS(vAxis := LIFT2)
    Frame (301,3 298x468)
        shows vAXIS(vAxis := XY2)
    Textfield (137,270 48x16), "%d", text variable: iOFFSET2
        OnMouseDown: write the text variable via Default
    Label (135,249 59x22), "OFFSET"
    Button (312,110 87x34), "STOP !!"
        OnMouseDown: execute { ACTION1.bSTOP_ALL:=TRUE; }
    Button (11,111 87x33), "STOP !!"
        OnMouseDown: execute { ACTION1.bSTOP_ALL:=TRUE; }
    Button (54,272 73x19), "SET"
        tap bWP_Start
END_VISUALIZATION

// ---- POUs/AXES/vAXIS.TcVIS
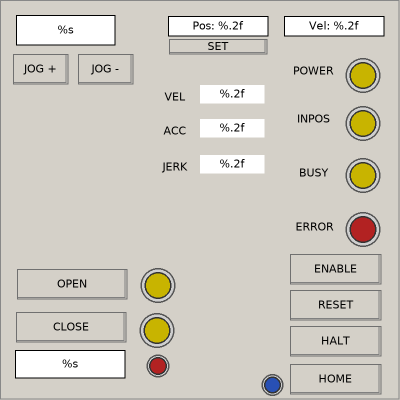
VISUALIZATION vAXIS  // 400x400
VAR_IN_OUT
	vAxis:FB_Axis;
END_VAR
    Rectangle (168,16 100x20), "Pos: %.2f", text variable: vAxis.rActPos
    Rectangle (284,16 100x20), "Vel: %.2f", text variable: vAxis.rActVel
    Lamp1 (343,53 40x45), variable: vAxis.power.Enable, style: Lamp-Lamp1-Yellow
    Label (286,60 55x22), "POWER"
    Lamp1 (343,101 40x45), variable: vAxis.bInPos, style: Lamp-Lamp1-Yellow
    Lamp1 (343,207 40x45), variable: vAxis.bAXIS_ERROR, style: Lamp-Lamp1-Red
    Lamp1 (343,153 40x45), variable: vAxis.bBusy, style: Lamp-Lamp1-Yellow
    Label (286,108 55x22), "INPOS"
    Label (287,216 55x22), "ERROR"
    Label (286,162 55x22), "BUSY"
    Button (290,254 91x30), "ENABLE"
        toggle vAxis.bEnable
    Button (290,290 91x30), "RESET"
        toggle vAxis.bReset
    Button (290,326 91x30), "HALT"
        tap vAxis.bHalt
    Textfield (199,84 66x20), "%.2f", text variable: vAxis.rVel
        OnMouseDown: write the text variable via Default
    Label (157,86 36x22), "VEL"
    Textfield (199,154 66x20), "%.2f", text variable: vAxis.rJerk
        OnMouseDown: write the text variable via Default
    Label (157,156 36x22), "JERK"
    Textfield (199,118 66x20), "%.2f", text variable: vAxis.rAcc
        OnMouseDown: write the text variable via Default
    Label (157,120 36x22), "ACC"
    Button (13,54 55x30), "JOG +"
        tap vAxis.bJogPos
    Button (78,54 55x30), "JOG -"
        tap vAxis.bJogNeg
    Rectangle (16,15 99x30), "%s", text variable: vAxis.sName
    Button (169,39 98x15), "SET"
        tap vAxis.bSetPosition
    Button (17,269 110x30), "OPEN"
        OnMouseDown: execute { vAXIS.bOPEN:=TRUE;  vAXIS.bCLOSE:=FALSE; }
    Button (16,312 110x30), "CLOSE"
        OnMouseDown: execute { vAXIS.bCLOSE:=TRUE; vAXIS.bOPEN:=FALSE; }
    Lamp1 (138,263 40x45), variable: vAxis.bLIMIT_OPENED, style: Lamp-Lamp1-Yellow
    Lamp1 (137,308 40x45), variable: vAxis.bLIMIT_CLOSED, style: Lamp-Lamp1-Yellow
    Rectangle (15,350 110x28), "%s", text variable: vAxis.sAXIS_STATE
    Button (290,364 91x30), "HOME"
        OnMouseDown: execute { vAxis.bHOME:=TRUE; }
    Lamp1 (260,368 25x34), variable: vAxis.bHOMED, style: Lamp-Lamp1-Blue
    Lamp1 (145,352 26x28), variable: vAxis.bSTATE_ERROR, style: Lamp-Lamp1-Red
END_VISUALIZATION

// ---- POUs/AXES/vAXES1.TcVIS
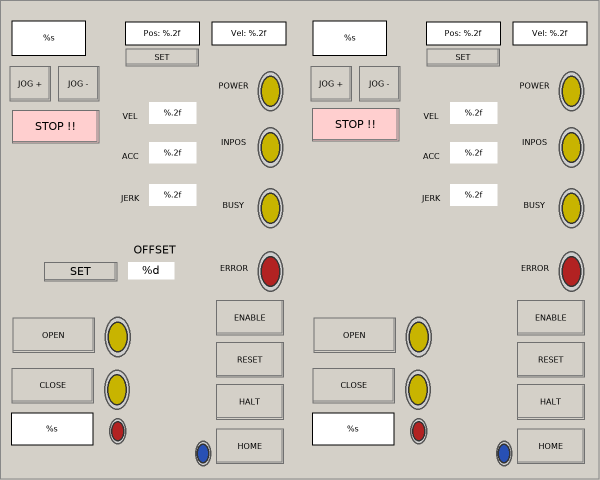
VISUALIZATION vAXES1  // 600x480
    Frame (0,3 298x468)
        shows vAXIS(vAxis := LIFT1)
    Frame (301,3 298x468)
        shows vAXIS(vAxis := XY1)
    Textfield (127,261 48x19), "%d", text variable: iOFFSET1
        OnMouseDown: write the text variable via Default
    Label (125,239 59x22), "OFFSET"
    Button (12,110 87x33), "STOP !!"
        OnMouseDown: execute { ACTION1.bSTOP_ALL:=TRUE; }
    Button (312,108 87x33), "STOP !!"
        OnMouseDown: execute { ACTION1.bSTOP_ALL:=TRUE; }
    Button (44,262 73x19), "SET"
        tap bWP_Start
END_VISUALIZATION

// ---- POUs/EVENT_LOGGER/vEVENT_LOGGER.TcVIS
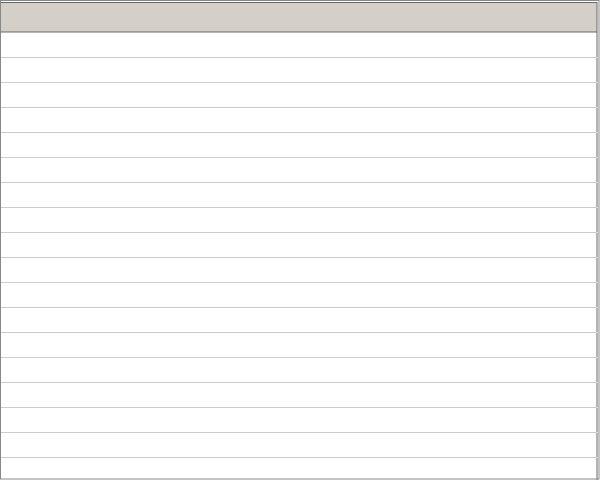
VISUALIZATION vEVENT_LOGGER  // 600x480
    Table (-3,2 600x480), data array: fbEventLogger.EventBuffer
        p3854506369: fbEventLogger.EventBuffer[INDEX].eEventType
        p1892666644: fbEventLogger.EventBuffer[INDEX].eEventSeverity
        p338671338: fbEventLogger.EventBuffer[INDEX].nEventIdentity
        p2170511999: fbEventLogger.EventBuffer[INDEX].sEventName
        p3723444502: fbEventLogger.EventBuffer[INDEX].sEventText
        p1218418051: fbEventLogger.EventBuffer[INDEX].dtTimestamp
END_VISUALIZATION

// ---- POUs/PISTONS/vPISTONS.TcVIS
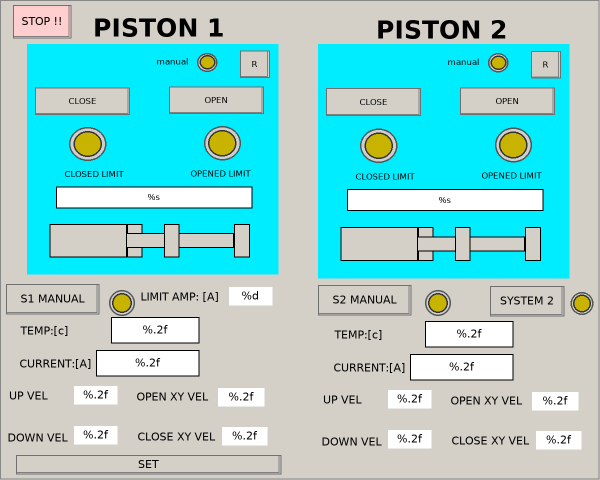
VISUALIZATION vPISTONS  // 600x480
    Frame (318,44 251x234), invisible if: true
        shows vPISTON(PIST1 := PIST2, MANUAL := ACTION2.bMANUAL)
    Frame (27,44 251x230)
        shows vPISTON(PIST1 := PIST1, MANUAL := ACTION1.bMANUAL)
    Label (84,14 150x27), "PISTON 1"
    Label (367,16 150x27), "PISTON 2", invisible if: true
    Button (490,286 74x30), "SYSTEM 2", invisible if: true
        toggle bSECOND_SYS
    Label (-17,385 91x22), "UP VEL"
    Label (-8,427 91x22), "DOWN VEL"
    Textfield (73,425 45x20), "%.2f", text variable: LIFT1_DOWN_VEL
        OnMouseDown: write the text variable via Default
    Textfield (217,387 48x20), "%.2f", text variable: XY1_OPEN_VEL
        OnMouseDown: write the text variable via Default
    Label (127,386 91x22), "OPEN XY VEL"
    Textfield (221,426 47x20), "%.2f", text variable: XY1_CLOSE_VEL
        OnMouseDown: write the text variable via Default
    Label (131,426 91x22), "CLOSE XY VEL"
    Label (77,297 91x22)
    Label (358,297 91x22)
    Rectangle (111,317 88x26), "%.2f", text variable: ACTION1.iTEMP_SHOW
    Rectangle (96,350 103x26), "%.2f", text variable: ACTION1.iCURRENT_PISTON_SHOW
    Label (18,320 53x22), "TEMP:[c]"
    Label (10,353 91x22), "CURRENT:[A]"
    Button (6,284 93x30), "S1 MANUAL"
        OnMouseDown: execute { ACTION1.bMANUAL:=TRUE; }
    Lamp1 (107,285 30x36), variable: ACTION1.bMANUAL, style: Lamp-Lamp1-Yellow
    Button (318,285 93x30), "S2 MANUAL", invisible if: true, input disabled if: NOT ACTION2.bALL_HOMED
        OnMouseDown: execute { ACTION2.bMANUAL:=TRUE; }
    Lamp1 (423,285 30x36), variable: ACTION2.bMANUAL, invisible if: true, style: Lamp-Lamp1-Yellow
    Lamp1 (569,288 26x31), variable: bSECOND_SYS, invisible if: true, style: Lamp-Lamp1-Yellow
    Button (13,5 58x33), "STOP !!"
        OnMouseDown: execute { ACTION1.bSTOP_ALL:=TRUE; }
    Textfield (73,385 45x20), "%.2f", text variable: LIFT1_UP_VEL
        OnMouseDown: write the text variable via Default
    Button (16,455 265x19), "SET"
        tap bWP_Start
    Label (138,286 84x22), "LIMIT AMP: [A]"
    Textfield (228,286 45x20), "%d", text variable: SAFETY_LIMIT1
        OnMouseDown: write the text variable via Default
    Label (297,389 91x22), "UP VEL", invisible if: true
    Label (306,431 91x22), "DOWN VEL", invisible if: true
    Textfield (387,429 45x20), "%.2f", text variable: LIFT2_DOWN_VEL, invisible if: true
        OnMouseDown: write the text variable via Default
    Textfield (531,391 48x20), "%.2f", text variable: XY2_OPEN_VEL, invisible if: true
        OnMouseDown: write the text variable via Default
    Label (441,390 91x22), "OPEN XY VEL", invisible if: true
    Textfield (535,430 47x20), "%.2f", text variable: XY2_CLOSE_VEL, invisible if: true
        OnMouseDown: write the text variable via Default
    Label (445,430 91x22), "CLOSE XY VEL", invisible if: true
    Rectangle (425,321 88x26), "%.2f", text variable: ACTION1.iTEMP_SHOW, invisible if: true
    Rectangle (410,354 103x26), "%.2f", text variable: ACTION1.iCURRENT_PISTON_SHOW, invisible if: true
    Label (332,324 53x22), "TEMP:[c]", invisible if: true
    Label (324,357 91x22), "CURRENT:[A]", invisible if: true
    Textfield (387,389 45x20), "%.2f", text variable: LIFT2_UP_VEL, invisible if: true
        OnMouseDown: write the text variable via Default
END_VISUALIZATION

// ---- POUs/PISTONS/vPISTON.TcVIS
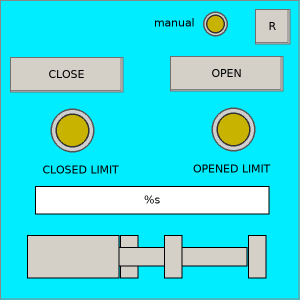
VISUALIZATION vPISTON  // 300x300
VAR_IN_OUT
	PIST1: FB_PISTON;
	MANUAL:BOOL;
	
END_VAR
    Button (170,56 113x35), "OPEN"
        OnMouseDown: execute { PIST1.bOPEN_CMD:=TRUE; }
    Rectangle (35,186 234x28), "%s", text variable: PIST1.sSTATE
    Lamp1 (47,104 51x53), variable: PIST1.bCLOSED_LIMIT, style: Lamp-Lamp1-Yellow
    Label (31,155 99x30), "CLOSED LIMIT"
    Lamp1 (208,103 51x53), variable: PIST1.bOPEN_LIMIT, style: Lamp-Lamp1-Yellow
    Label (182,154 99x30), "OPENED LIMIT"
    Button (10,57 113x35), "CLOSE"
        OnMouseDown: execute { PIST1.bOPEN_CMD:=FALSE; }
    Lamp1 (200,10 31x28), variable: PIST1.bLOCAL_MANUAL, style: Lamp-Lamp1-Yellow
    Button (255,9 35x35), "R", colour toggle: PIST1.bLOCAL_MANUAL
        tap PIST1.bLOCAL_RESET
    Rectangle (119,247 128x19), invisible if: NOT PIST1.bOPENED
    Rectangle (248,235 18x43), invisible if: NOT PIST1.bOPENED
    Rectangle (120,235 18x43), invisible if: NOT PIST1.bCLOSED
    Rectangle (78,247 92x19), invisible if: NOT PIST1.bBUSY
    Rectangle (164,235 18x43), invisible if: NOT PIST1.bBUSY
    Rectangle (27,235 92x43), colour toggle: PIST1.bERROR
    Label (125,8 99x30), "manual"
END_VISUALIZATION

// ---- VISUs/VISUs/vCOMM.TcVIS
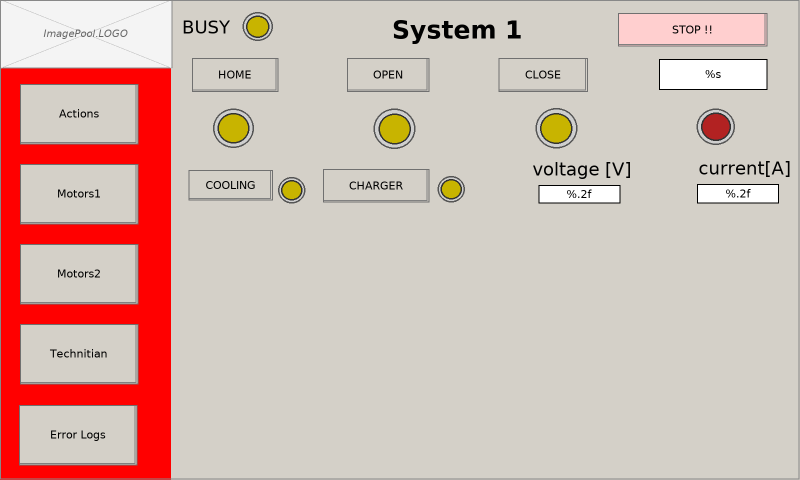
VISUALIZATION vCOMM  // 800x480
    Button (20,84 118x60), "Actions"
        OnMouseClick: FrameSelectionChange Selection=SelectedFrame=c79d80b7-c479-4a39-9ec5-d387b8e1dbac, GlobSel=AssignType=Directly, SelType=Locally
    Button (20,164 118x60), "Motors1", input disabled if: NOT ACTION1.bMANUAL
        OnMouseClick: FrameSelectionChange Selection=SelectedFrame=c79d80b7-c479-4a39-9ec5-d387b8e1dbac, Selection=1, GlobSel=AssignType=Directly, SelType=Locally
    Button (20,244 118x60), "Motors2", input disabled if: NOT ACTION2.bMANUAL
        OnMouseClick: FrameSelectionChange Selection=SelectedFrame=c79d80b7-c479-4a39-9ec5-d387b8e1dbac, Selection=2, GlobSel=AssignType=Directly, SelType=Locally
    Button (19,405 118x60), "Error Logs"
        OnMouseClick: FrameSelectionChange Selection=SelectedFrame=c79d80b7-c479-4a39-9ec5-d387b8e1dbac, Selection=3, GlobSel=AssignType=Directly, SelType=Locally
    Frame (171,-1 630x483)
        shows vACTION(vACTION := ACTION1, vACTION2 := ACTION2)
        shows vAXES1()
        shows vAXES2()
        shows vEVENT_LOGGER()
        shows vPISTONS()
    Button (20,324 118x60), "Technitian"
        OnMouseClick: FrameSelectionChange Selection=SelectedFrame=c79d80b7-c479-4a39-9ec5-d387b8e1dbac, Selection=4, GlobSel=AssignType=Directly, SelType=Locally
    Image (0,-1 172x69), image: ImagePool.LOGO
END_VISUALIZATION

// ---- VISUs/VISUs/vMAIN.TcVIS
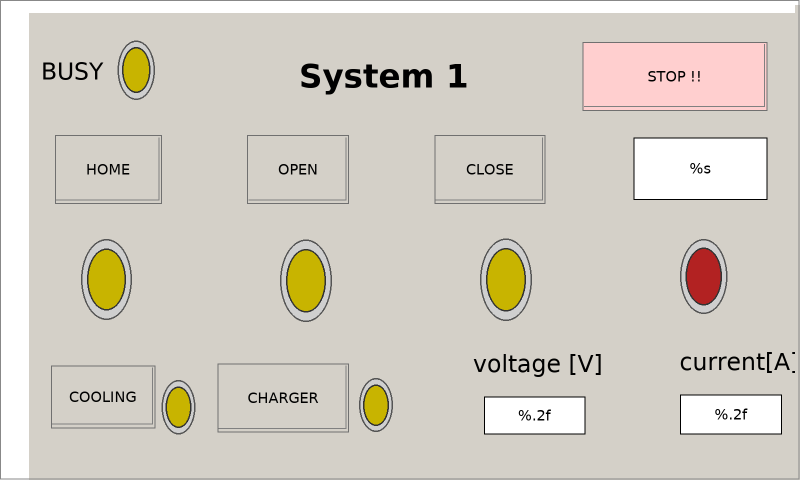
VISUALIZATION vMAIN  // 800x480
    Frame (29,13 780x996)
        shows vACTION(vACTION := ACTION1, vACTION2 := ACTION2)
    Frame (795,5 780x1000)
        shows vACTION(vACTION := ACTION1, vACTION2 := ACTION2)
    Table (37,1012 1084x201), data array: fbEventLogger.EventBuffer
        p3854506369: fbEventLogger.EventBuffer[INDEX].eEventType
        p1892666644: fbEventLogger.EventBuffer[INDEX].eEventSeverity
        p338671338: fbEventLogger.EventBuffer[INDEX].nEventIdentity
        p2170511999: fbEventLogger.EventBuffer[INDEX].sEventName
        p3723444502: fbEventLogger.EventBuffer[INDEX].sEventText
        p1218418051: fbEventLogger.EventBuffer[INDEX].dtTimestamp
END_VISUALIZATION
